TYPE FLOWMETER_VALUES :
STRUCT
	MassFlow:REAL;
	VolumeFlow:REAL;
	CorrectedVolueFLow:REAL;
	Density:REAL;
	ReferenceDensity:REAL;
	Temperature:REAL;
	TotalMass:REAL;
END_STRUCT
END_TYPE

(* stored: Version 1.1.0.1, ProductVersion 3.1.0.26
   DUT FLOWMETER_VALUES: Id {a013a2b7-ddda-4b28-8464-000384e35c04} *)
